RoboDK station: main for aircraft (copy).rdk

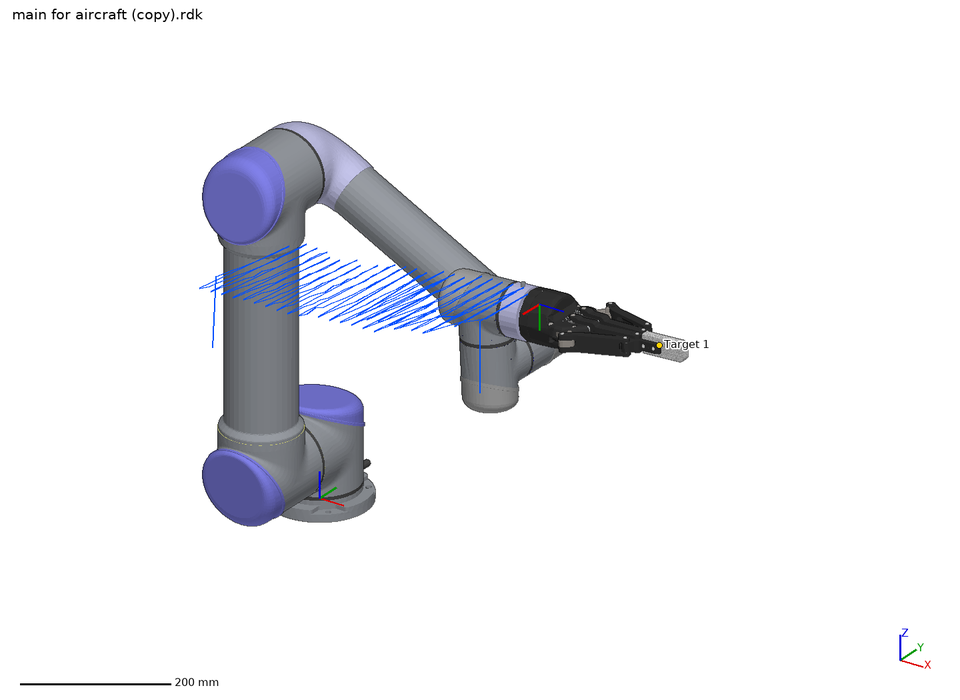
[picture v0: the station drawn from its stored meshes, robots at their saved joint values, targets as dots, program paths as lines]
Station main. Poses are relative to the parent item; angles as X-Y-Z fixed-axis rotations.
  - frame UR5 Base at (0, 0, 0) mm
    - robot UR5: 6 axes, payload 5 kg, reach 850 mm, repeatability 0.1 mm, weight 18.4 kg
        modified DH rows (alpha deg, a mm, theta deg, d mm): 0, 0, 0, 89.2; 90, 0, 180, 0; 0, 425, 0, 0; 0, 392.43, 0, 109; -90, 0, 0, 93.65; 90, 0, 180, 82
        joint limits [-360, -360, -360, -360, -360, -360] to [360, 360, 360, 360, 360, 360]; home [0, -90, -90, 0, 90, 0]; saved at [-0.013, -90.021, -116.97, 29.935, 90.025, 0.152]
      - tool RobotiQ 2-Finger-140 Closed, TCP at (0, 0, 200) mm, size 124 x 75 x 244.3 mm
    - target Target 1 (Cartesian target) at (626.33, -109, 443.99) mm, rotated rx -87.03 ry 0 rz -90 deg; joints [0, -90, -117.03, 30, 90, 0] of UR5
  - frame Object at (435.27, -113.47, 453.26) mm, rotated rx -90 ry 0 rz -90 deg
    - object cloud_1 at (0, 0, 0) mm
  - machining project Path1 settings: rotZ(0) | rotX(0)*rotY(0) | rotz(0) | onStart | onPathStart | onApproach | onPoint | onRetract | onFinish | SetRPM(%1) | SetTool(%1) | Extruder(%1) | default | default | OutOnMov(%1) | OutOffMov(%1) | onPathFinish | M_RunCode(%1)
  - program Path1 (311 instructions, listed below)
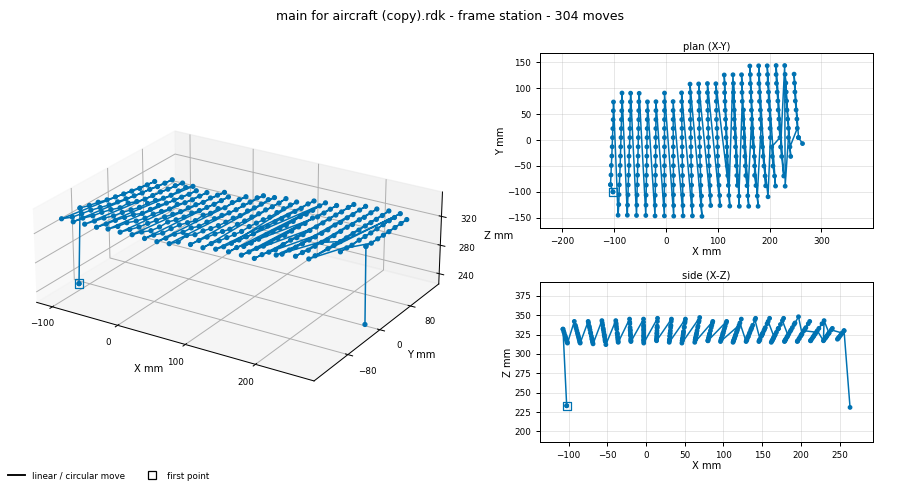
[picture p0: tool path of main for aircraft (copy).rdk in frame station, 304 of 304 moves have a stored position in this frame; points joined in program order, loops and branches not executed]

--- program Path1 (robot UR5) ---
  Smooth(10)
  Set Ref.: UR5 Base
  Set Tool: RobotiQ 2-Finger-140 Closed
  Show RobotiQ 2-Finger-140 Closed
  Set speed (1000.0 mm/s)
  MoveJ 1 to (-102.38, -99.99, 233.07) mm, rotated rx 0 ry 8.41 rz 109.19 deg; joints [12.602, -85.858, -96.132, -6.063, 80.274, 110.751]
  MoveL 2 to (-102.38, -99.99, 233.07) mm, rotated rx 0 ry 8.41 rz 109.19 deg; joints [12.602, -85.858, -96.132, -6.063, 80.274, 110.751]
  MoveL 3 to (-107.19, -86.18, 332) mm, rotated rx 0 ry 8.41 rz 109.19 deg; joints [10.562, -99.693, -83.593, -4.724, 82.295, 110.463]
  MoveL 4 to (-107.19, -86.18, 332) mm, rotated rx 0 ry 8.41 rz 109.19 deg; joints [10.562, -99.693, -83.593, -4.724, 82.295, 110.463]
  Set speed (25.0 mm/s)
  MoveL 5 to (-106.22, -67.34, 329) mm, rotated rx 0 ry 8.74 rz 104.18 deg; joints [10.87, -99.349, -86.354, -2.871, 81.384, 105.634]
  MoveL 6 to (-105.57, -48.98, 327) mm, rotated rx 0 ry 8.16 rz 105.57 deg; joints [10.82, -99.525, -89.316, 0.897, 81.464, 106.907]
  MoveL 7 to (-104.6, -30.75, 324) mm, rotated rx 0 ry 7.53 rz 107.19 deg; joints [10.76, -99.737, -92.273, 4.74, 81.545, 108.407]
  MoveL 8 to (-103.96, -12.89, 322) mm, rotated rx 0 ry 7.37 rz 117.72 deg; joints [10.016, -100.321, -94.773, 8.532, 83.469, 118.664]
  MoveL 9 to (-103.31, 4.75, 320) mm, rotated rx 0 ry 7.46 rz 117.73 deg; joints [9.953, -100.71, -96.926, 10.993, 83.577, 118.674]
  MoveL 10 to (-102.67, 22.18, 318) mm, rotated rx 0 ry 7.52 rz 128.57 deg; joints [9.186, -101.609, -99.093, 14.811, 85.544, 129.274]
  MoveL 11 to (-102.02, 39.38, 316) mm, rotated rx 0 ry 6.96 rz 132.96 deg; joints [9.121, -102.574, -101.234, 18.709, 85.65, 133.56]
  MoveL 12 to (-101.7, 56.55, 315) mm, rotated rx 0 ry 6.41 rz 138.18 deg; joints [9.085, -103.834, -103.068, 22.622, 85.712, 138.679]
  MoveL 13 to (-101.37, 73.6, 314) mm, rotated rx 0 ry 3.46 rz 132.88 deg; joints [10.558, -105.526, -105.133, 28.096, 81.808, 133.3]
  MoveL 14 to (-92.54, -145.08, 342) mm, rotated rx 0 ry 12.08 rz 94.29 deg; joints [9.643, -101.198, -70.072, -20.918, 81.468, 96.221]
  MoveL 15 to (-91.18, -124.47, 337) mm, rotated rx 0 ry 10.91 rz 107.25 deg; joints [8.275, -100.357, -75.36, -14.733, 85.077, 108.45]
  MoveL 16 to (-90.64, -105.34, 335) mm, rotated rx 0 ry 8.32 rz 121.32 deg; joints [7.646, -100.444, -80.524, -6.143, 86.725, 121.995]
  MoveL 17 to (-90.1, -86.44, 333) mm, rotated rx 0 ry 8.35 rz 111.38 deg; joints [8.357, -100.028, -83.281, -4.497, 84.755, 112.306]
  MoveL 18 to (-89.29, -67.55, 330) mm, rotated rx 0 ry 9.44 rz 103.06 deg; joints [8.831, -99.489, -85.62, -4.149, 83.408, 104.309]
  MoveL 19 to (-88.48, -48.98, 327) mm, rotated rx 0 ry 7.86 rz 110.36 deg; joints [8.456, -99.825, -89.329, 1.751, 84.342, 111.271]
  MoveL 20 to (-87.94, -30.85, 325) mm, rotated rx 0 ry 7.28 rz 107.7 deg; joints [8.741, -100.08, -92.048, 5.148, 83.531, 108.625]
  MoveL 21 to (-87.4, -12.93, 323) mm, rotated rx 0 ry 8.39 rz 105.46 deg; joints [8.687, -100.038, -93.905, 5.809, 83.628, 106.526]
  MoveL 22 to (-86.86, 4.77, 321) mm, rotated rx 0 ry 6.63 rz 99.81 deg; joints [9.338, -100.841, -96.822, 11.062, 81.85, 100.818]
  MoveL 23 to (-86.31, 22.25, 319) mm, rotated rx 0 ry 5.26 rz 109.06 deg; joints [8.973, -102.005, -99.329, 16.325, 82.775, 109.764]
  MoveL 24 to (-86.04, 39.63, 318) mm, rotated rx 0 ry 5.54 rz 114.92 deg; joints [8.583, -102.815, -101.017, 18.776, 83.783, 115.571]
  MoveL 25 to (-85.5, 56.73, 316) mm, rotated rx 0 ry 5.08 rz 117.6 deg; joints [8.547, -103.81, -102.937, 22.22, 83.831, 118.178]
  MoveL 26 to (-85.23, 73.83, 315) mm, rotated rx 0 ry 3.41 rz 99.66 deg; joints [9.627, -105.263, -104.828, 26.693, 80.961, 100.21]
  MoveL 27 to (-84.96, 90.83, 314) mm, rotated rx 0 ry 3.94 rz 89.7 deg; joints [9.971, -106.042, -106.185, 28.226, 80.032, 90.395]
  MoveL 28 to (-74.66, -145.08, 342) mm, rotated rx 0 ry 10.54 rz 100.52 deg; joints [7.023, -101.454, -71.046, -17.903, 85.006, 101.612]
  MoveL 29 to (-74.22, -125.57, 340) mm, rotated rx 0 ry 9.71 rz 108.2 deg; joints [6.378, -101.067, -75.24, -12.926, 86.723, 108.974]
  MoveL 30 to (-73.35, -105.66, 336) mm, rotated rx 0 ry 8.84 rz 106.92 deg; joints [6.599, -100.447, -79.464, -8.567, 86.038, 107.705]
  MoveL 31 to (-72.91, -86.7, 334) mm, rotated rx 0 ry 8.21 rz 101.06 deg; joints [7.161, -100.199, -82.829, -5.067, 84.48, 101.952]
  MoveL 32 to (-72.26, -67.75, 331) mm, rotated rx 0 ry 9.2 rz 96.58 deg; joints [7.42, -99.749, -85.325, -4.123, 83.725, 97.683]
  MoveL 33 to (-71.39, -48.98, 327) mm, rotated rx 0 ry 7.88 rz 97.73 deg; joints [7.389, -99.789, -89.038, 0.969, 83.737, 98.667]
  MoveL 34 to (-71.39, -31.04, 327) mm, rotated rx 0 ry 6.46 rz 99.7 deg; joints [7.385, -100.613, -91.81, 6.015, 83.747, 100.462]
  MoveL 35 to (-70.51, -12.93, 323) mm, rotated rx 0 ry 7.59 rz 98.3 deg; joints [7.329, -100.32, -94.011, 6.781, 83.826, 99.186]
  MoveL 36 to (-69.86, 4.75, 320) mm, rotated rx 0 ry 7.15 rz 99.07 deg; joints [7.281, -100.728, -96.551, 10.182, 83.898, 99.896]
  MoveL 37 to (-69.64, 22.25, 319) mm, rotated rx 0 ry 5.47 rz 89.8 deg; joints [7.973, -101.873, -99.092, 15.437, 82.044, 90.568]
  MoveL 38 to (-69.42, 39.63, 318) mm, rotated rx 0 ry 4.41 rz 89.88 deg; joints [7.965, -103.107, -101.143, 19.794, 82.05, 90.502]
  MoveL 39 to (-68.98, 56.73, 316) mm, rotated rx 0 ry 3.93 rz 98.35 deg; joints [7.596, -104.158, -102.988, 23.224, 82.992, 98.85]
  MoveL 40 to (-68.77, 73.83, 315) mm, rotated rx 0 ry 5.61 rz 89.69 deg; joints [7.94, -104.282, -104.219, 22.835, 82.068, 90.473]
  MoveL 41 to (-68.33, 90.54, 313) mm, rotated rx 0 ry 5.55 rz 74.23 deg; joints [8.823, -105.26, -105.973, 25.806, 79.709, 75.129]
  MoveL 42 to (-56.95, -145.51, 343) mm, rotated rx 0 ry 9.64 rz 101.74 deg; joints [4.945, -101.92, -71.114, -16.416, 87.075, 102.389]
  MoveL 43 to (-56.45, -125.57, 340) mm, rotated rx 0 ry 8.37 rz 100.44 deg; joints [5.18, -101.276, -75.726, -11.245, 86.385, 101.075]
  MoveL 44 to (-55.95, -105.97, 337) mm, rotated rx 0 ry 8.97 rz 99.84 deg; joints [5.141, -100.723, -78.806, -9.321, 86.447, 100.511]
  MoveL 45 to (-55.29, -86.44, 333) mm, rotated rx 0 ry 8.77 rz 103.79 deg; joints [4.782, -100.34, -82.357, -5.829, 87.353, 104.341]
  MoveL 46 to (-54.96, -67.75, 331) mm, rotated rx 0 ry 10.15 rz 95.9 deg; joints [5.361, -99.868, -84.468, -5.787, 85.759, 96.747]
  MoveL 47 to (-54.46, -49.13, 328) mm, rotated rx 0 ry 8.29 rz 89.76 deg; joints [5.984, -99.98, -88.428, 0.073, 84.044, 90.628]
  MoveL 48 to (-53.96, -30.85, 325) mm, rotated rx 0 ry 5.34 rz 95.68 deg; joints [5.649, -100.888, -92.308, 7.865, 84.903, 96.178]
  MoveL 49 to (-53.8, -12.97, 324) mm, rotated rx 0 ry 7.69 rz 102.43 deg; joints [4.957, -100.783, -93.45, 6.716, 86.735, 102.97]
  MoveL 50 to (-53.46, 4.78, 322) mm, rotated rx 0 ry 8.12 rz 110.5 deg; joints [4.228, -101.283, -95.457, 9.135, 88.645, 110.872]
  MoveL 51 to (-52.97, 22.25, 319) mm, rotated rx 0 ry 6.28 rz 105.85 deg; joints [4.88, -102.068, -98.402, 14.419, 86.859, 106.271]
  MoveL 52 to (-52.63, 39.51, 317) mm, rotated rx 0 ry 5.01 rz 96.55 deg; joints [5.559, -103.021, -100.779, 18.808, 85.033, 97.01]
  MoveL 53 to (-52.63, 56.9, 317) mm, rotated rx 0 ry 3.88 rz 89.83 deg; joints [5.917, -104.494, -102.589, 23.18, 84.085, 90.228]
  MoveL 54 to (-52.47, 74.07, 316) mm, rotated rx 0 ry 6.25 rz 89.29 deg; joints [5.936, -104.353, -103.631, 21.699, 84.022, 89.941]
  MoveL 55 to (-51.8, 90.26, 312) mm, rotated rx 0 ry 6.86 rz 83.81 deg; joints [6.305, -104.639, -105.472, 23.236, 83.002, 84.609]
  MoveL 56 to (-39.02, -145.51, 343) mm, rotated rx 0 ry 10.41 rz 100.77 deg; joints [2.876, -102.295, -70.06, -17.872, 89.105, 101.109]
  MoveL 57 to (-38.68, -125.57, 340) mm, rotated rx 0 ry 8.6 rz 107.1 deg; joints [2.527, -101.795, -75.104, -11.321, 90.02, 107.285]
  MoveL 58 to (-38.45, -106.28, 338) mm, rotated rx 0 ry 9.51 rz 102.38 deg; joints [2.79, -101.253, -77.786, -10.244, 89.276, 102.667]
  MoveL 59 to (-38.11, -86.96, 335) mm, rotated rx 0 ry 10.02 rz 98.86 deg; joints [3.049, -100.721, -80.786, -8.4, 88.533, 99.253]
  MoveL 60 to (-37.77, -67.95, 332) mm, rotated rx 0 ry 8.81 rz 100.35 deg; joints [3.01, -100.662, -84.566, -3.438, 88.601, 100.688]
  MoveL 61 to (-37.2, -48.98, 327) mm, rotated rx 0 ry 8.58 rz 104.58 deg; joints [2.636, -100.453, -87.878, 0.03, 89.545, 104.809]
  MoveL 62 to (-37.09, -30.94, 326) mm, rotated rx 0 ry 6.73 rz 109.13 deg; joints [2.605, -101.258, -91.051, 5.948, 89.613, 109.295]
  MoveL 63 to (-36.97, -13.01, 325) mm, rotated rx 0 ry 5.81 rz 112.71 deg; joints [2.578, -102.029, -93.568, 10.238, 89.673, 112.841]
  MoveL 64 to (-36.63, 4.78, 322) mm, rotated rx 0 ry 7.75 rz 102.62 deg; joints [2.874, -101.51, -95.208, 9.15, 88.841, 102.888]
  MoveL 65 to (-36.4, 22.32, 320) mm, rotated rx 0 ry 8.53 rz 105.62 deg; joints [2.497, -101.848, -96.972, 10.603, 89.819, 105.812]
  MoveL 66 to (-36.18, 39.63, 318) mm, rotated rx 0 ry 5.1 rz 103.06 deg; joints [3.176, -103.547, -100.132, 18.704, 87.988, 103.282]
  MoveL 67 to (-35.95, 56.73, 316) mm, rotated rx 0 ry 3.37 rz 99.81 deg; joints [3.515, -104.997, -102.361, 24.03, 87.065, 100.001]
  MoveL 68 to (-35.84, 73.83, 315) mm, rotated rx 0 ry 6.51 rz 97.07 deg; joints [3.362, -104.518, -103.198, 21.245, 87.46, 97.408]
  MoveL 69 to (-21.21, -146.36, 345) mm, rotated rx 0 ry 10.78 rz 100.32 deg; joints [0.831, -103.07, -68.684, -18.857, 91.104, 100.296]
  MoveL 70 to (-20.97, -125.94, 341) mm, rotated rx 0 ry 9.17 rz 96.23 deg; joints [1.341, -102.102, -74.004, -13.009, 89.667, 96.363]
  MoveL 71 to (-20.85, -106.6, 339) mm, rotated rx 0 ry 8.79 rz 89.96 deg; joints [1.903, -101.608, -77.676, -9.513, 88.113, 90.252]
  MoveL 72 to (-20.54, -86.7, 334) mm, rotated rx 0 ry 9.41 rz 86.82 deg; joints [2.181, -100.816, -81.091, -7.498, 87.329, 87.221]
  MoveL 73 to (-20.35, -67.75, 331) mm, rotated rx 0 ry 8.78 rz 100.37 deg; joints [0.958, -100.98, -84.233, -3.424, 90.627, 100.391]
  MoveL 74 to (-20.29, -49.43, 330) mm, rotated rx 0 ry 8.07 rz 105.51 deg; joints [0.619, -101.412, -87.053, 0.689, 91.538, 105.446]
  MoveL 75 to (-20.11, -31.04, 327) mm, rotated rx 0 ry 7.55 rz 102.54 deg; joints [0.903, -101.463, -90.018, 4.108, 90.74, 102.548]
  MoveL 76 to (-19.92, -12.97, 324) mm, rotated rx 0 ry 5.89 rz 95.38 deg; joints [1.529, -101.925, -93.313, 9.371, 89.03, 95.508]
  MoveL 77 to (-19.92, 4.81, 324) mm, rotated rx 0 ry 6.5 rz 94.93 deg; joints [1.525, -102.397, -94.965, 10.889, 89.042, 95.07]
  MoveL 78 to (-19.68, 22.32, 320) mm, rotated rx 0 ry 8.26 rz 97.94 deg; joints [1.159, -102.119, -96.662, 10.596, 89.991, 98.024]
  MoveL 79 to (-19.55, 39.63, 318) mm, rotated rx 0 ry 5.79 rz 107.49 deg; joints [0.794, -103.81, -99.357, 17.649, 90.946, 107.486]
  MoveL 80 to (-19.49, 56.9, 317) mm, rotated rx 0 ry 4.26 rz 114.24 deg; joints [0.782, -105.413, -101.378, 22.905, 90.968, 114.234]
  MoveL 81 to (-19.43, 74.07, 316) mm, rotated rx 0 ry 6.19 rz 111.98 deg; joints [0.436, -105.6, -102.418, 22.278, 91.878, 111.909]
  MoveL 82 to (-3.18, -146.36, 345) mm, rotated rx 0 ry 10.73 rz 100.34 deg; joints [-1.217, -103.634, -68.014, -18.926, 93.112, 99.939]
  MoveL 83 to (-3.14, -125.94, 341) mm, rotated rx 0 ry 11.27 rz 87.5 deg; joints [0.124, -102.309, -72.137, -16.813, 89.389, 87.57]
  MoveL 84 to (-3.11, -105.97, 337) mm, rotated rx 0 ry 10.22 rz 84.32 deg; joints [0.416, -101.559, -76.799, -11.811, 88.584, 84.481]
  MoveL 85 to (-3.09, -86.96, 335) mm, rotated rx 0 ry 7.59 rz 89.98 deg; joints [-0.16, -101.783, -81.227, -4.58, 90.156, 89.964]
  MoveL 86 to (-3.06, -67.95, 332) mm, rotated rx 0 ry 6.84 rz 103.6 deg; joints [-1.091, -102.038, -84.402, -0.215, 92.689, 103.379]
  MoveL 87 to (-3.04, -49.43, 330) mm, rotated rx 0 ry 8.39 rz 101.11 deg; joints [-1.099, -101.741, -86.307, -0.189, 92.699, 100.838]
  MoveL 88 to (-3.02, -31.04, 327) mm, rotated rx 0 ry 8.41 rz 97.48 deg; joints [-0.808, -101.633, -89.075, 2.362, 91.892, 97.288]
  MoveL 89 to (-2.99, -12.97, 324) mm, rotated rx 0 ry 5.88 rz 95.42 deg; joints [-0.504, -102.411, -92.718, 9.27, 91.056, 95.345]
  MoveL 90 to (-2.98, 4.8, 323) mm, rotated rx 0 ry 6.56 rz 99.89 deg; joints [-0.84, -102.841, -94.416, 10.789, 91.959, 99.728]
  MoveL 91 to (-2.96, 22.39, 321) mm, rotated rx 0 ry 8.19 rz 93.99 deg; joints [-0.516, -102.65, -96.025, 10.506, 91.08, 93.88]
  MoveL 92 to (-2.93, 39.63, 318) mm, rotated rx 0 ry 5.24 rz 109.31 deg; joints [-1.217, -104.536, -98.879, 18.461, 92.944, 109.132]
  MoveL 93 to (-2.93, 57.08, 318) mm, rotated rx 0 ry 3.75 rz 117.73 deg; joints [-1.224, -106.292, -100.706, 23.678, 92.964, 117.61]
  MoveL 94 to (-2.91, 74.07, 316) mm, rotated rx 0 ry 6.01 rz 107.04 deg; joints [-1.238, -105.986, -101.901, 22.137, 92.989, 106.829]
  MoveL 95 to (-2.9, 90.83, 314) mm, rotated rx 0 ry 8.15 rz 102.6 deg; joints [-1.251, -105.83, -103.026, 20.892, 93.012, 102.305]
  MoveL 96 to (14.9, -146.78, 346) mm, rotated rx 0 ry 10.58 rz 92.62 deg; joints [-2.457, -104.157, -67.286, -19.135, 92.897, 92.127]
  MoveL 97 to (14.72, -126.31, 342) mm, rotated rx 0 ry 12.07 rz 92.33 deg; joints [-2.453, -103.205, -70.364, -18.509, 92.886, 91.762]
  MoveL 98 to (14.46, -105.66, 336) mm, rotated rx 0 ry 9.79 rz 96.03 deg; joints [-2.767, -102.37, -76.175, -11.209, 93.75, 95.474]
  MoveL 99 to (14.38, -86.7, 334) mm, rotated rx 0 ry 5.33 rz 107.43 deg; joints [-3.109, -103.006, -81.616, -0.482, 94.692, 107.084]
  MoveL 100 to (14.38, -68.36, 334) mm, rotated rx 0 ry 7.78 rz 101.88 deg; joints [-3.102, -102.698, -82.806, -2.135, 94.671, 101.358]
  MoveL 101 to (14.21, -49.43, 330) mm, rotated rx 0 ry 10.19 rz 93.02 deg; joints [-2.489, -101.744, -84.835, -3.612, 92.983, 92.529]
  MoveL 102 to (14.08, -31.04, 327) mm, rotated rx 0 ry 6.92 rz 99.29 deg; joints [-2.837, -102.609, -89.019, 4.782, 93.932, 98.889]
  MoveL 103 to (14.03, -13.05, 326) mm, rotated rx 0 ry 5.97 rz 100.93 deg; joints [-2.85, -103.327, -91.556, 9.006, 93.966, 100.585]
  MoveL 104 to (13.91, 4.8, 323) mm, rotated rx 0 ry 7.02 rz 113.7 deg; joints [-3.826, -103.748, -93.3, 10.576, 96.619, 113.114]
  MoveL 105 to (13.82, 22.39, 321) mm, rotated rx 0 ry 7.7 rz 98.65 deg; joints [-2.862, -103.489, -95.404, 11.26, 93.991, 98.193]
  MoveL 106 to (13.73, 39.76, 319) mm, rotated rx 0 ry 5.75 rz 107.77 deg; joints [-3.221, -105.003, -97.866, 17.369, 94.961, 107.382]
  MoveL 107 to (13.69, 57.08, 318) mm, rotated rx 0 ry 2.98 rz 112.99 deg; joints [-2.883, -107.001, -100.217, 24.465, 94.045, 112.829]
  MoveL 108 to (13.65, 74.3, 317) mm, rotated rx 0 ry 6.62 rz 105.49 deg; joints [-3.227, -106.368, -100.895, 20.859, 94.971, 105.028]
  MoveL 109 to (32.89, -146.36, 345) mm, rotated rx 0 ry 10.2 rz 84.56 deg; joints [-3.687, -104.429, -67.314, -18.421, 92.668, 83.997]
  MoveL 110 to (32.6, -126.31, 342) mm, rotated rx 0 ry 10.93 rz 97.86 deg; joints [-5.021, -104.126, -70.137, -16.631, 96.418, 96.776]
  MoveL 111 to (32.12, -105.97, 337) mm, rotated rx 0 ry 10.44 rz 104.05 deg; joints [-5.594, -103.496, -74.436, -12.293, 98.027, 102.836]
  MoveL 112 to (32.03, -87.21, 336) mm, rotated rx 0 ry 6.19 rz 115.52 deg; joints [-5.706, -104.098, -79.801, -1.745, 98.342, 114.83]
  MoveL 113 to (31.84, -68.36, 334) mm, rotated rx 0 ry 8.14 rz 90.15 deg; joints [-4.215, -102.954, -82.094, -3.115, 94.194, 89.555]
  MoveL 114 to (31.46, -49.43, 330) mm, rotated rx 0 ry 10.66 rz 90.09 deg; joints [-4.184, -102.205, -83.905, -4.578, 94.128, 89.311]
  MoveL 115 to (31.07, -30.94, 326) mm, rotated rx 0 ry 5.28 rz 90.17 deg; joints [-4.205, -103.361, -89.271, 7.34, 94.203, 89.78]
  MoveL 116 to (31.17, -13.09, 327) mm, rotated rx 0 ry 5.96 rz 100.94 deg; joints [-4.841, -104.101, -90.583, 8.806, 95.944, 100.391]
  MoveL 117 to (30.79, 4.8, 323) mm, rotated rx 0 ry 7.52 rz 94.41 deg; joints [-4.51, -103.579, -92.684, 8.734, 95.047, 93.779]
  MoveL 118 to (30.79, 22.53, 323) mm, rotated rx 0 ry 7.63 rz 94.41 deg; joints [-4.514, -104.263, -94.441, 11.066, 95.059, 93.771]
  MoveL 119 to (30.31, 39.63, 318) mm, rotated rx 0 ry 4.96 rz 97.03 deg; joints [-4.531, -105.491, -97.649, 18.192, 95.121, 96.615]
  MoveL 120 to (30.41, 57.26, 319) mm, rotated rx 0 ry 2.81 rz 102.12 deg; joints [-4.529, -107.619, -99.406, 24.271, 95.112, 101.892]
  MoveL 121 to (30.22, 74.3, 317) mm, rotated rx 0 ry 5.15 rz 108.57 deg; joints [-5.128, -107.635, -100.424, 23.145, 96.747, 108.059]
  MoveL 122 to (30.03, 91.12, 315) mm, rotated rx 0 ry 5.56 rz 104.8 deg; joints [-4.997, -108.236, -101.985, 24.81, 96.393, 104.259]
  MoveL 123 to (50.92, -146.36, 345) mm, rotated rx 0 ry 11.06 rz 97.54 deg; joints [-6.983, -105.741, -65.013, -20.323, 98.297, 96.066]
  MoveL 124 to (50.48, -126.31, 342) mm, rotated rx 0 ry 8.95 rz 113.5 deg; joints [-8.14, -105.608, -70.208, -12.561, 101.613, 112.059]
  MoveL 125 to (50.18, -106.91, 340) mm, rotated rx 0 ry 9.24 rz 106.56 deg; joints [-7.631, -104.869, -73.51, -10.617, 100.162, 105.167]
  MoveL 126 to (49.44, -86.96, 335) mm, rotated rx 0 ry 9.48 rz 109.47 deg; joints [-7.906, -104.284, -77.111, -7.702, 100.955, 107.979]
  MoveL 127 to (49.3, -68.36, 334) mm, rotated rx 0 ry 9.07 rz 90.13 deg; joints [-6.19, -103.51, -80.707, -4.901, 96.133, 89.151]
  MoveL 128 to (48.56, -49.28, 329) mm, rotated rx 0 ry 10.66 rz 92.94 deg; joints [-6.443, -102.892, -83.087, -4.742, 96.874, 91.692]
  MoveL 129 to (48.41, -31.13, 328) mm, rotated rx 0 ry 5.83 rz 84.78 deg; joints [-5.878, -104.048, -87.973, 6.189, 95.318, 84.213]
  MoveL 130 to (48.12, -13.05, 326) mm, rotated rx 0 ry 5.33 rz 90.21 deg; joints [-6.182, -104.609, -90.334, 9.58, 96.174, 89.632]
  MoveL 131 to (47.82, 4.81, 324) mm, rotated rx 0 ry 7.2 rz 76.49 deg; joints [-5.193, -104.12, -92.385, 9.49, 93.476, 75.959]
  MoveL 132 to (47.38, 22.39, 321) mm, rotated rx 0 ry 7.14 rz 99.47 deg; joints [-6.803, -105.001, -93.912, 11.801, 97.924, 98.562]
  MoveL 133 to (47.08, 39.76, 319) mm, rotated rx 0 ry 4.41 rz 97.99 deg; joints [-6.495, -106.524, -96.747, 18.87, 97.088, 97.467]
  MoveL 134 to (47.08, 57.26, 319) mm, rotated rx 0 ry 4.01 rz 125.33 deg; joints [-7.472, -108.39, -97.913, 22.981, 99.779, 124.828]
  MoveL 135 to (46.79, 74.3, 317) mm, rotated rx 0 ry 4.5 rz 121.3 deg; joints [-7.475, -108.943, -99.475, 24.517, 99.794, 120.718]
  MoveL 136 to (46.79, 91.7, 317) mm, rotated rx 0 ry 6.11 rz 121.36 deg; joints [-7.941, -109.626, -100.266, 24.578, 101.082, 120.479]
  MoveL 137 to (46.34, 108.07, 314) mm, rotated rx 0 ry 10.92 rz 117.12 deg; joints [-8.885, -108.695, -100.471, 19.168, 103.71, 115.154]
  MoveL 138 to (69.35, -147.2, 347) mm, rotated rx 0 ry 12 rz 99.79 deg; joints [-9.237, -107.157, -62.368, -22.52, 101.064, 97.663]
  MoveL 139 to (68.15, -125.94, 341) mm, rotated rx 0 ry 7.89 rz 98 deg; joints [-8.776, -105.727, -70.4, -11.805, 99.788, 96.716]
  MoveL 140 to (68.55, -107.86, 343) mm, rotated rx 0 ry 8.48 rz 97.55 deg; joints [-8.787, -105.837, -72.46, -10.235, 99.802, 96.168]
  MoveL 141 to (67.15, -87.21, 336) mm, rotated rx 0 ry 10.36 rz 95.98 deg; joints [-8.708, -104.568, -75.681, -10.205, 99.64, 94.313]
  MoveL 142 to (66.75, -68.36, 334) mm, rotated rx 0 ry 9.61 rz 99.51 deg; joints [-8.982, -104.614, -79.001, -6.02, 100.437, 97.877]
  MoveL 143 to (65.96, -49.43, 330) mm, rotated rx 0 ry 10.69 rz 87.23 deg; joints [-7.801, -103.571, -82.191, -5, 97.153, 85.83]
  MoveL 144 to (65.36, -31.04, 327) mm, rotated rx 0 ry 6.34 rz 85.26 deg; joints [-7.823, -104.524, -86.994, 5.147, 97.253, 84.424]
  MoveL 145 to (64.96, -13.01, 325) mm, rotated rx 0 ry 4.93 rz 77.04 deg; joints [-7.493, -105.162, -90.026, 10.35, 96.361, 76.456]
  MoveL 146 to (64.76, 4.81, 324) mm, rotated rx 0 ry 6.51 rz 100.09 deg; joints [-8.728, -105.642, -90.876, 10.01, 99.812, 99.041]
  MoveL 147 to (64.16, 22.39, 321) mm, rotated rx 0 ry 6.34 rz 111.08 deg; joints [-9.349, -106.434, -92.917, 13.312, 101.575, 109.985]
  MoveL 148 to (64.16, 40, 321) mm, rotated rx 0 ry 4.74 rz 127.04 deg; joints [-9.682, -108.313, -94.835, 19.275, 102.513, 126.291]
  MoveL 149 to (63.76, 57.26, 319) mm, rotated rx 0 ry 4.94 rz 117.85 deg; joints [-9.37, -108.619, -96.702, 20.86, 101.649, 117.032]
  MoveL 150 to (63.56, 74.54, 318) mm, rotated rx 0 ry 3.5 rz 109.62 deg; joints [-8.739, -109.8, -98.764, 25.22, 99.899, 109.083]
  MoveL 151 to (63.56, 91.99, 318) mm, rotated rx 0 ry 4.51 rz 121.63 deg; joints [-9.402, -110.978, -99.543, 26.596, 101.746, 120.908]
  MoveL 152 to (62.96, 108.41, 315) mm, rotated rx 0 ry 7.19 rz 112.07 deg; joints [-9.55, -110.437, -100.692, 24.312, 102.18, 110.779]
  MoveL 153 to (86.23, -126.31, 342) mm, rotated rx 0 ry 9.23 rz 87.58 deg; joints [-9.907, -106.325, -68.517, -14.504, 99.39, 86.01]
  MoveL 154 to (85.73, -106.91, 340) mm, rotated rx 0 ry 8.04 rz 83.22 deg; joints [-9.609, -105.849, -72.899, -9.328, 98.569, 81.939]
  MoveL 155 to (84.97, -87.47, 337) mm, rotated rx 0 ry 11.02 rz 79.42 deg; joints [-8.967, -104.812, -74.94, -11.158, 96.794, 77.915]
  MoveL 156 to (84.21, -68.36, 334) mm, rotated rx 0 ry 9.54 rz 86.91 deg; joints [-9.768, -104.966, -78.512, -6.174, 99.12, 85.324]
  MoveL 157 to (83.2, -49.43, 330) mm, rotated rx 0 ry 10.68 rz 87.2 deg; joints [-9.71, -104.409, -81.138, -5.255, 99.022, 85.435]
  MoveL 158 to (82.2, -30.94, 326) mm, rotated rx 0 ry 6.38 rz 100.32 deg; joints [-10.641, -105.636, -85.603, 4.824, 101.718, 99.078]
  MoveL 159 to (82.2, -13.05, 326) mm, rotated rx 0 ry 4.07 rz 114.45 deg; joints [-10.957, -107.168, -88.228, 11.6, 102.617, 113.674]
  MoveL 160 to (81.69, 4.81, 324) mm, rotated rx 0 ry 6.45 rz 115.59 deg; joints [-11.516, -107.114, -89.394, 10.509, 104.236, 114.256]
  MoveL 161 to (81.44, 22.53, 323) mm, rotated rx 0 ry 6.04 rz 101.08 deg; joints [-10.632, -107.237, -91.86, 13.044, 101.733, 99.9]
  MoveL 162 to (80.94, 40, 321) mm, rotated rx 0 ry 4.5 rz 105.14 deg; joints [-10.641, -108.452, -94.195, 18.21, 101.785, 104.278]
  MoveL 163 to (80.68, 57.44, 320) mm, rotated rx 0 ry 3.88 rz 98.82 deg; joints [-10.319, -109.369, -96.124, 21.587, 100.89, 98.097]
  MoveL 164 to (80.18, 74.54, 318) mm, rotated rx 0 ry 3.49 rz 109.56 deg; joints [-10.624, -110.562, -97.682, 24.884, 101.774, 108.904]
  MoveL 165 to (79.93, 91.7, 317) mm, rotated rx 0 ry 4.04 rz 107.19 deg; joints [-10.627, -111.304, -99.005, 26.365, 101.796, 106.425]
  MoveL 166 to (79.93, 109.1, 317) mm, rotated rx 0 ry 5.62 rz 99.39 deg; joints [-10.459, -111.611, -100.069, 26.021, 101.325, 98.319]
  MoveL 167 to (104.11, -126.31, 342) mm, rotated rx 0 ry 10.94 rz 100.97 deg; joints [-13.037, -107.98, -65.179, -17.951, 104.871, 98.279]
  MoveL 168 to (103.5, -106.91, 340) mm, rotated rx 0 ry 9.27 rz 99.63 deg; joints [-12.788, -107.383, -70.024, -12.017, 104.166, 97.434]
  MoveL 169 to (102.28, -87.21, 336) mm, rotated rx 0 ry 9.33 rz 90.07 deg; joints [-11.956, -106.273, -74.217, -9.042, 101.807, 88.107]
  MoveL 170 to (101.37, -68.16, 333) mm, rotated rx 0 ry 9.49 rz 93.26 deg; joints [-12.199, -106.038, -77.195, -6.476, 102.567, 91.173]
  MoveL 171 to (100.45, -49.43, 330) mm, rotated rx 0 ry 10.2 rz 99.03 deg; joints [-12.712, -105.992, -79.546, -4.85, 104.105, 96.619]
  MoveL 172 to (99.54, -31.04, 327) mm, rotated rx 0 ry 5.74 rz 125.49 deg; joints [-13.675, -107.821, -83.922, 6.86, 106.955, 124.198]
  MoveL 173 to (99.54, -13.09, 327) mm, rotated rx 0 ry 4.97 rz 132.47 deg; joints [-13.696, -108.728, -86.154, 11.054, 107.017, 131.458]
  MoveL 174 to (98.93, 4.83, 325) mm, rotated rx 0 ry 6.9 rz 113.84 deg; joints [-13.359, -107.994, -87.831, 9.256, 106.06, 112.169]
  MoveL 175 to (98.32, 22.53, 323) mm, rotated rx 0 ry 6.13 rz 106.2 deg; joints [-12.783, -108.274, -90.488, 12.68, 104.422, 104.766]
  MoveL 176 to (97.41, 39.88, 320) mm, rotated rx 0 ry 5.55 rz 102.18 deg; joints [-12.475, -108.717, -92.953, 16.091, 103.586, 100.919]
  MoveL 177 to (97.41, 57.44, 320) mm, rotated rx 0 ry 3.99 rz 107.03 deg; joints [-12.49, -110.353, -94.753, 21.177, 103.631, 106.146]
  MoveL 178 to (97.11, 74.77, 319) mm, rotated rx 0 ry 4.46 rz 97.66 deg; joints [-12.165, -110.834, -96.397, 22.702, 102.722, 96.682]
  MoveL 179 to (96.8, 91.99, 318) mm, rotated rx 0 ry 3.37 rz 100.37 deg; joints [-12.171, -112.38, -97.941, 26.926, 102.756, 99.638]
  MoveL 180 to (96.19, 108.76, 316) mm, rotated rx 0 ry 3.39 rz 85.16 deg; joints [-11.662, -113.085, -99.707, 29.348, 101.356, 84.474]
  MoveL 181 to (120.2, -87.47, 337) mm, rotated rx 0 ry 11.39 rz 105.6 deg; joints [-15.3, -108.21, -70.373, -12.959, 108.052, 102.274]
  MoveL 182 to (119.13, -68.36, 334) mm, rotated rx 0 ry 8.68 rz 103.94 deg; joints [-14.852, -107.855, -75.561, -5.379, 106.769, 101.537]
  MoveL 183 to (118.06, -49.58, 331) mm, rotated rx 0 ry 8.38 rz 116.28 deg; joints [-15.651, -108.359, -78.321, -1.27, 109.209, 113.895]
  MoveL 184 to (116.99, -31.13, 328) mm, rotated rx 0 ry 5.99 rz 129.64 deg; joints [-15.731, -109.161, -82.141, 6.411, 109.496, 128.161]
  MoveL 185 to (117.35, -13.17, 329) mm, rotated rx 0 ry 6.18 rz 122.8 deg; joints [-15.494, -109.48, -83.951, 7.947, 108.77, 121.18]
  MoveL 186 to (115.92, 4.83, 325) mm, rotated rx 0 ry 7.5 rz 98.76 deg; joints [-14.298, -108.114, -86.823, 7.253, 105.314, 96.792]
  MoveL 187 to (115.56, 22.6, 324) mm, rotated rx 0 ry 6.64 rz 104.97 deg; joints [-14.6, -109.163, -88.875, 11.362, 106.217, 103.195]
  MoveL 188 to (114.85, 40.13, 322) mm, rotated rx 0 ry 4.87 rz 118.31 deg; joints [-14.916, -110.711, -91.114, 17.337, 107.18, 117.068]
  MoveL 189 to (114.14, 57.44, 320) mm, rotated rx 0 ry 4.43 rz 121.51 deg; joints [-14.904, -111.592, -93.019, 20.662, 107.183, 120.421]
  MoveL 190 to (113.78, 74.77, 319) mm, rotated rx 0 ry 5.09 rz 103.56 deg; joints [-14.296, -111.615, -94.835, 21.32, 105.432, 102.239]
  MoveL 191 to (113.07, 91.7, 317) mm, rotated rx 0 ry 3.5 rz 109.84 deg; joints [-14.288, -113.241, -96.629, 26.455, 105.451, 108.962]
  MoveL 192 to (113.07, 109.1, 317) mm, rotated rx 0 ry 4.26 rz 114.74 deg; joints [-14.595, -114.318, -97.475, 27.766, 106.341, 113.667]
  MoveL 193 to (112.35, 125.7, 315) mm, rotated rx 0 ry 7.55 rz 117.68 deg; joints [-15.435, -114.292, -97.909, 25.136, 108.827, 115.597]
  MoveL 194 to (123.05, -127.42, 345) mm, rotated rx 0 ry 11.81 rz 113.8 deg; joints [-16.182, -110.57, -61.425, -19.552, 110.617, 110.137]
  MoveL 195 to (121.27, -106.91, 340) mm, rotated rx 0 ry 11.54 rz 112.57 deg; joints [-15.993, -109.32, -66.269, -15.757, 110.107, 109.046]
  MoveL 196 to (129.23, 126.1, 316) mm, rotated rx 0 ry 5.68 rz 99.25 deg; joints [-15.877, -115.167, -97.586, 26.898, 106.71, 97.609]
  MoveL 197 to (137.82, -87.47, 337) mm, rotated rx 0 ry 11.64 rz 100.27 deg; joints [-16.58, -108.988, -68.958, -14.124, 108.298, 96.638]
  MoveL 198 to (136.59, -68.36, 334) mm, rotated rx 0 ry 9.05 rz 100.11 deg; joints [-16.378, -108.715, -74.038, -6.602, 107.755, 97.363]
  MoveL 199 to (135.77, -49.73, 332) mm, rotated rx 0 ry 6.81 rz 103.97 deg; joints [-16.429, -109.141, -77.917, 0.108, 107.957, 101.918]
  MoveL 200 to (135.36, -31.42, 331) mm, rotated rx 0 ry 5.77 rz 96.28 deg; joints [-15.925, -109.29, -81.076, 4.382, 106.474, 94.613]
  MoveL 201 to (134.14, -13.13, 328) mm, rotated rx 0 ry 6.36 rz 95.8 deg; joints [-15.883, -109.175, -83.515, 6.096, 106.425, 93.966]
  MoveL 202 to (133.32, 4.84, 326) mm, rotated rx 0 ry 6.4 rz 90.57 deg; joints [-15.561, -109.279, -86.018, 8.652, 105.525, 88.79]
  MoveL 203 to (132.09, 22.53, 323) mm, rotated rx 0 ry 5.59 rz 107.75 deg; joints [-16.373, -110.422, -87.967, 12.792, 108.002, 106.099]
  MoveL 204 to (131.68, 40.13, 322) mm, rotated rx 0 ry 4.65 rz 137.21 deg; joints [-17.243, -112.537, -89.394, 18.557, 110.627, 136.114]
  MoveL 205 to (131.68, 57.8, 322) mm, rotated rx 0 ry 6.11 rz 118.91 deg; joints [-16.989, -112.347, -90.716, 17.375, 109.863, 117.114]
  MoveL 206 to (130.46, 74.77, 319) mm, rotated rx 0 ry 7.67 rz 112.69 deg; joints [-16.928, -112.121, -92.349, 16.954, 109.744, 110.322]
  MoveL 207 to (130.05, 91.99, 318) mm, rotated rx 0 ry 2.81 rz 102.37 deg; joints [-15.773, -114.406, -95.386, 26.931, 106.356, 101.576]
  MoveL 208 to (130.05, 109.44, 318) mm, rotated rx 0 ry 3.52 rz 109.9 deg; joints [-16.076, -115.489, -96.216, 28.242, 107.245, 108.905]
  MoveL 209 to (141.5, -127.79, 346) mm, rotated rx 0 ry 10.32 rz 93.34 deg; joints [-16.004, -110.526, -61.821, -18.394, 106.336, 90.337]
  MoveL 210 to (140.68, -108.17, 344) mm, rotated rx 0 ry 11.45 rz 102.65 deg; joints [-16.871, -110.479, -64.107, -17.234, 109.029, 98.999]
  MoveL 211 to (147.13, 74.77, 319) mm, rotated rx 0 ry 6.65 rz 96.13 deg; joints [-17.53, -112.637, -91.979, 17.657, 108.118, 93.998]
  MoveL 212 to (146.67, 91.99, 318) mm, rotated rx 0 ry 3.35 rz 100.46 deg; joints [-17.51, -115.073, -93.907, 25.509, 108.089, 99.399]
  MoveL 213 to (146.21, 109.1, 317) mm, rotated rx 0 ry 3.37 rz 100.47 deg; joints [-17.497, -116.096, -95.205, 27.811, 108.079, 99.399]
  MoveL 214 to (145.75, 126.1, 316) mm, rotated rx 0 ry 3.75 rz 88.77 deg; joints [-17.123, -116.782, -96.691, 29.551, 107.005, 87.619]
  MoveL 215 to (156.35, -87.99, 339) mm, rotated rx 0 ry 13.38 rz 88.06 deg; joints [-17.078, -109.569, -66.643, -17.722, 106.153, 84.058]
  MoveL 216 to (154.05, -68.36, 334) mm, rotated rx 0 ry 8.55 rz 94.22 deg; joints [-17.668, -109.633, -73.076, -6.267, 108.093, 91.462]
  MoveL 217 to (153.13, -49.73, 332) mm, rotated rx 0 ry 4.18 rz 98.06 deg; joints [-17.695, -110.605, -77.758, 4.009, 108.232, 96.72]
  MoveL 218 to (152.2, -31.32, 330) mm, rotated rx 0 ry 7.3 rz 99.02 deg; joints [-17.891, -110.007, -78.999, 1.389, 108.884, 96.609]
  MoveL 219 to (150.82, -13.09, 327) mm, rotated rx 0 ry 8.39 rz 90.43 deg; joints [-17.29, -109.325, -81.736, 2.274, 107.162, 87.822]
  MoveL 220 to (150.36, 4.84, 326) mm, rotated rx 0 ry 5.87 rz 90.49 deg; joints [-17.317, -110.509, -84.728, 9.091, 107.274, 88.66]
  MoveL 221 to (149.9, 22.67, 325) mm, rotated rx 0 ry 5.39 rz 90.53 deg; joints [-17.309, -111.226, -86.808, 12.388, 107.28, 88.846]
  MoveL 222 to (148.97, 40.25, 323) mm, rotated rx 0 ry 2.68 rz 92.94 deg; joints [-17.353, -112.896, -89.271, 19.358, 107.471, 92.103]
  MoveL 223 to (149.44, 58.16, 324) mm, rotated rx 0 ry 4.9 rz 92 deg; joints [-17.362, -113.005, -90.18, 18.05, 107.467, 90.462]
  MoveL 224 to (159.58, -127.79, 346) mm, rotated rx 0 ry 9.43 rz 90.48 deg; joints [-17.551, -111.667, -60.894, -17.322, 107.384, 87.502]
  MoveL 225 to (157.74, -107.54, 342) mm, rotated rx 0 ry 11.34 rz 90.34 deg; joints [-17.437, -110.555, -63.965, -17.357, 107.153, 86.799]
  MoveL 226 to (165.34, 40.13, 322) mm, rotated rx 0 ry 3.98 rz 55.89 deg; joints [-17.854, -112.831, -88.859, 18.266, 105.591, 54.904]
  MoveL 227 to (164.83, 57.62, 321) mm, rotated rx 0 ry 5.23 rz 72.13 deg; joints [-18.135, -113.042, -89.979, 17.832, 106.462, 70.587]
  MoveL 228 to (164.32, 75.01, 320) mm, rotated rx 0 ry 6.12 rz 85.86 deg; joints [-18.68, -113.694, -90.883, 18.158, 108.13, 83.828]
  MoveL 229 to (163.8, 92.28, 319) mm, rotated rx 0 ry 3.91 rz 99.04 deg; joints [-19.219, -115.945, -92.149, 23.988, 109.787, 97.671]
  MoveL 230 to (162.78, 109.1, 317) mm, rotated rx 0 ry 3.51 rz 109.84 deg; joints [-19.475, -117.249, -93.412, 27.136, 110.631, 108.635]
  MoveL 231 to (162.78, 126.5, 317) mm, rotated rx 0 ry 2.79 rz 111.34 deg; joints [-19.395, -118.817, -94.506, 30.556, 110.387, 110.4]
  MoveL 232 to (161.75, 142.99, 315) mm, rotated rx 0 ry 5.34 rz 113.35 deg; joints [-19.874, -118.873, -95.271, 28.86, 111.911, 111.463]
  MoveL 233 to (173.56, -87.73, 338) mm, rotated rx 0 ry 12.03 rz 108.38 deg; joints [-20.799, -112.333, -64.304, -15.878, 114.124, 103.577]
  MoveL 234 to (170.99, -68.16, 333) mm, rotated rx 0 ry 9.46 rz 112.83 deg; joints [-20.768, -111.782, -69.983, -7.788, 114.164, 109.166]
  MoveL 235 to (170.99, -49.88, 333) mm, rotated rx 0 ry 7.09 rz 122.31 deg; joints [-20.889, -112.621, -73.518, -0.45, 114.551, 119.765]
  MoveL 236 to (170.48, -31.51, 332) mm, rotated rx 0 ry 8.03 rz 109.51 deg; joints [-20.333, -111.943, -75.998, -0.268, 112.817, 106.482]
  MoveL 237 to (168.43, -13.13, 328) mm, rotated rx 0 ry 8.43 rz 101.46 deg; joints [-19.79, -111.182, -79.259, 1.575, 111.243, 98.349]
  MoveL 238 to (166.89, 4.83, 325) mm, rotated rx 0 ry 5.87 rz 96.02 deg; joints [-19.288, -111.661, -83.129, 8.586, 109.798, 93.941]
  MoveL 239 to (166.37, 22.6, 324) mm, rotated rx 0 ry 5.56 rz 78.42 deg; joints [-18.428, -111.785, -85.963, 12.05, 107.229, 76.671]
  MoveL 240 to (177.67, -127.79, 346) mm, rotated rx 0 ry 10.14 rz 125.61 deg; joints [-21.909, -115.54, -56.206, -17.547, 117.545, 121.711]
  MoveL 241 to (176.13, -107.86, 343) mm, rotated rx 0 ry 11.44 rz 113.11 deg; joints [-21.198, -113.812, -59.923, -17.907, 115.277, 108.498]
  MoveL 242 to (183.31, 22.6, 324) mm, rotated rx 0 ry 5.24 rz 115.3 deg; joints [-21.707, -114.31, -82.859, 11.99, 113.864, 113.295]
  MoveL 243 to (182.18, 40.13, 322) mm, rotated rx 0 ry 4.63 rz 127.23 deg; joints [-21.949, -115.404, -84.759, 16.107, 114.699, 125.621]
  MoveL 244 to (182.18, 57.8, 322) mm, rotated rx 0 ry 5.34 rz 115.88 deg; joints [-21.716, -115.612, -86.327, 16.68, 113.964, 113.84]
  MoveL 245 to (180.48, 74.77, 319) mm, rotated rx 0 ry 4.67 rz 112.45 deg; joints [-21.419, -116.117, -88.655, 20.078, 113.137, 110.673]
  MoveL 246 to (180.48, 92.28, 319) mm, rotated rx 0 ry 4.46 rz 98.37 deg; joints [-20.88, -116.738, -90.471, 22.472, 111.463, 96.659]
  MoveL 247 to (179.35, 109.1, 317) mm, rotated rx 0 ry 3.92 rz 99.61 deg; joints [-20.853, -117.817, -92.036, 25.703, 111.457, 98.115]
  MoveL 248 to (179.35, 126.5, 317) mm, rotated rx 0 ry 2.28 rz 105.51 deg; joints [-20.849, -119.906, -93.069, 30.611, 111.443, 104.657]
  MoveL 249 to (178.78, 143.44, 316) mm, rotated rx 0 ry 4.57 rz 101.36 deg; joints [-20.945, -119.884, -94.068, 29.127, 111.777, 99.604]
  MoveL 250 to (192.36, -88.25, 340) mm, rotated rx 0 ry 14.31 rz 118.57 deg; joints [-23.679, -115.36, -58.963, -20.17, 119.83, 112.012]
  MoveL 251 to (191.23, -69.18, 338) mm, rotated rx 0 ry 10.5 rz 121.78 deg; joints [-23.252, -114.723, -65.469, -9.953, 118.445, 117.34]
  MoveL 252 to (188.97, -50.03, 334) mm, rotated rx 0 ry 8.34 rz 117.24 deg; joints [-22.51, -113.757, -70.803, -3.699, 116.113, 113.834]
  MoveL 253 to (187.27, -31.42, 331) mm, rotated rx 0 ry 7.3 rz 102.92 deg; joints [-21.494, -112.784, -75.16, 0.215, 112.946, 99.991]
  MoveL 254 to (186.14, -13.17, 329) mm, rotated rx 0 ry 9.38 rz 100.13 deg; joints [-21.413, -112.288, -76.948, -0.786, 112.762, 96.354]
  MoveL 255 to (184.44, 4.84, 326) mm, rotated rx 0 ry 7.61 rz 107.06 deg; joints [-21.685, -113.077, -80.003, 5.128, 113.726, 103.986]
  MoveL 256 to (196.89, -109.43, 348) mm, rotated rx 0 ry 8.54 rz 102.79 deg; joints [-21.844, -115.311, -59.185, -14.586, 113.482, 99.287]
  MoveL 257 to (201.48, 4.84, 326) mm, rotated rx 0 ry 7.7 rz 110.81 deg; joints [-23.502, -114.548, -77.926, 4.457, 116.03, 107.442]
  MoveL 258 to (200.86, 22.67, 325) mm, rotated rx 0 ry 5.99 rz 129.41 deg; joints [-24.007, -116.339, -79.94, 11.053, 117.72, 127.128]
  MoveL 259 to (200.24, 40.38, 324) mm, rotated rx 0 ry 4.92 rz 132.26 deg; joints [-23.791, -117.136, -82.215, 15.261, 117.047, 130.5]
  MoveL 260 to (199.63, 57.98, 323) mm, rotated rx 0 ry 6.53 rz 126.76 deg; joints [-24.009, -117.35, -83.376, 14.815, 117.801, 124.172]
  MoveL 261 to (197.77, 75.01, 320) mm, rotated rx 0 ry 5.59 rz 120.97 deg; joints [-23.514, -117.582, -86.054, 18.291, 116.298, 118.718]
  MoveL 262 to (197.77, 92.57, 320) mm, rotated rx 0 ry 5.64 rz 120.99 deg; joints [-23.526, -118.565, -87.308, 20.475, 116.337, 118.709]
  MoveL 263 to (195.92, 109.1, 317) mm, rotated rx 0 ry 4.57 rz 105.53 deg; joints [-22.715, -118.796, -90.022, 24.003, 113.865, 103.623]
  MoveL 264 to (195.92, 126.5, 317) mm, rotated rx 0 ry 2.01 rz 125.62 deg; joints [-22.719, -121.432, -91.032, 30.677, 113.879, 124.908]
  MoveL 265 to (195.3, 143.44, 316) mm, rotated rx 1.22 ry -0.93 rz -91.24 deg; joints [-22.716, -122.957, -92.016, 33.93, 113.911, 268.359]
  MoveL 266 to (211.37, -88.77, 342) mm, rotated rx 0 ry 12.2 rz 97.41 deg; joints [-23.104, -114.994, -59.803, -18.48, 114.117, 92.067]
  MoveL 267 to (209.51, -69.39, 339) mm, rotated rx 0 ry 10.52 rz 105.86 deg; joints [-23.686, -115.034, -64.083, -12.165, 116.146, 101.095]
  MoveL 268 to (206.42, -50.03, 334) mm, rotated rx 0 ry 10.07 rz 104.62 deg; joints [-23.475, -114.127, -68.51, -8.179, 115.639, 100.116]
  MoveL 269 to (205.19, -31.51, 332) mm, rotated rx 0 ry 7.38 rz 106.88 deg; joints [-23.346, -114.476, -72.748, -0.59, 115.293, 103.661]
  MoveL 270 to (203.95, -13.21, 330) mm, rotated rx 0 ry 8.53 rz 108.32 deg; joints [-23.52, -114.435, -74.721, 0.144, 115.938, 104.538]
  MoveL 271 to (219.86, 4.87, 328) mm, rotated rx 0 ry 7.08 rz 108.65 deg; joints [-24.889, -116.176, -75.906, 4.554, 116.963, 105.356]
  MoveL 272 to (218.52, 22.74, 326) mm, rotated rx 0 ry 4.28 rz 121.49 deg; joints [-24.898, -117.57, -78.842, 12.312, 117.078, 119.69]
  MoveL 273 to (217.85, 40.5, 325) mm, rotated rx 0 ry 5.06 rz 109.6 deg; joints [-24.628, -117.476, -80.841, 13.004, 116.23, 107.317]
  MoveL 274 to (216.51, 57.98, 323) mm, rotated rx 0 ry 5.62 rz 107.91 deg; joints [-24.592, -117.722, -82.714, 14.478, 116.2, 105.348]
  MoveL 275 to (215.84, 75.48, 322) mm, rotated rx 0 ry 4.64 rz 112.08 deg; joints [-24.598, -118.922, -84.439, 18.569, 116.265, 110.021]
  MoveL 276 to (214.5, 92.57, 320) mm, rotated rx 0 ry 5.88 rz 125.54 deg; joints [-25.279, -119.96, -85.138, 19.651, 118.595, 123.067]
  MoveL 277 to (213.16, 109.44, 318) mm, rotated rx 0 ry 5.65 rz 120.81 deg; joints [-25.017, -120.446, -87.043, 21.999, 117.812, 118.365]
  MoveL 278 to (212.49, 126.5, 317) mm, rotated rx 0 ry 3.93 rz 137.09 deg; joints [-25.021, -122.546, -88.276, 27.798, 117.868, 135.747]
  MoveL 279 to (212.49, 143.9, 317) mm, rotated rx 1.7 ry -0.97 rz -91.73 deg; joints [-24.499, -124.301, -89.714, 32.876, 116.162, 267.8]
  MoveL 280 to (227.23, -69.39, 339) mm, rotated rx 0 ry 10.15 rz 116.92 deg; joints [-25.972, -117.497, -61.238, -11.737, 120.185, 111.974]
  MoveL 281 to (223.21, -31.61, 333) mm, rotated rx 0 ry 9.64 rz 112.64 deg; joints [-25.522, -116.23, -68.766, -5.169, 118.878, 107.986]
  MoveL 282 to (221.2, -13.21, 330) mm, rotated rx 0 ry 8.83 rz 100.82 deg; joints [-24.611, -115.235, -73.113, -1.308, 115.959, 96.687]
  MoveL 283 to (229.06, 143.9, 317) mm, rotated rx 0 ry 2.37 rz 137.25 deg; joints [-26.03, -125.108, -87.8, 31.089, 117.76, 136.425]
  MoveL 284 to (229.92, -89.03, 343) mm, rotated rx 0 ry 10.45 rz 100.9 deg; joints [-24.931, -117.073, -58.089, -16.313, 116.464, 95.914]
  MoveL 285 to (236.28, 4.86, 327) mm, rotated rx 0 ry 7.18 rz 112.56 deg; joints [-26.579, -117.614, -73.803, 3.828, 119.129, 109.007]
  MoveL 286 to (236.28, 22.81, 327) mm, rotated rx 0 ry 5.19 rz 115.82 deg; joints [-26.417, -118.69, -76.35, 9.717, 118.58, 113.362]
  MoveL 287 to (234.84, 40.5, 325) mm, rotated rx 0 ry 5.54 rz 107.68 deg; joints [-26.122, -118.57, -78.758, 11.362, 117.682, 104.978]
  MoveL 288 to (233.39, 57.98, 323) mm, rotated rx 0 ry 5.49 rz 102.08 deg; joints [-25.851, -118.766, -81.077, 13.82, 116.876, 99.406]
  MoveL 289 to (232.67, 75.48, 322) mm, rotated rx 0 ry 4.47 rz 104.9 deg; joints [-25.849, -119.933, -82.822, 17.904, 116.918, 102.739]
  MoveL 290 to (231.95, 92.86, 321) mm, rotated rx 0 ry 4.66 rz 112.11 deg; joints [-26.087, -120.957, -83.964, 20.044, 117.757, 109.896]
  MoveL 291 to (231.22, 110.13, 320) mm, rotated rx 0 ry 5.15 rz 123.63 deg; joints [-26.534, -122.249, -84.68, 22.008, 119.304, 121.322]
  MoveL 292 to (229.78, 126.9, 318) mm, rotated rx 0 ry 4.3 rz 131.65 deg; joints [-26.513, -123.584, -86.136, 26.032, 119.325, 129.925]
  MoveL 293 to (240.62, -31.61, 333) mm, rotated rx 0 ry 10.88 rz 103.15 deg; joints [-26.452, -116.814, -66.6, -8.654, 118.417, 97.574]
  MoveL 294 to (239.17, -13.25, 331) mm, rotated rx 0 ry 8.01 rz 109.77 deg; joints [-26.612, -117.576, -70.485, -0.565, 119.059, 105.736]
  MoveL 295 to (253.38, 22.81, 327) mm, rotated rx 0 ry 6.33 rz 134.45 deg; joints [-28.74, -121.11, -72.696, 8.414, 123.069, 131.681]
  MoveL 296 to (252.6, 40.63, 326) mm, rotated rx 0 ry 5.94 rz 112.14 deg; joints [-27.829, -120.248, -75.996, 9.899, 119.921, 109.076]
  MoveL 297 to (251.05, 58.16, 324) mm, rotated rx 0 ry 6 rz 112.15 deg; joints [-27.796, -120.623, -78.045, 12.26, 119.908, 109.052]
  MoveL 298 to (249.5, 75.48, 322) mm, rotated rx 0 ry 4.21 rz 106.3 deg; joints [-27.336, -121.36, -80.764, 17.523, 118.443, 104.143]
  MoveL 299 to (248.73, 92.86, 321) mm, rotated rx 0 ry 3.3 rz 89.96 deg; joints [-26.822, -122.054, -83.006, 21.36, 116.772, 88.288]
  MoveL 300 to (247.95, 110.13, 320) mm, rotated rx 0 ry 4.27 rz 106.16 deg; joints [-27.294, -122.962, -83.657, 21.952, 118.405, 103.979]
  MoveL 301 to (247.18, 127.3, 319) mm, rotated rx 0 ry 4.69 rz 119.73 deg; joints [-27.745, -124.323, -84.228, 23.851, 119.99, 117.46]
  MoveL 302 to (255.7, 4.9, 330) mm, rotated rx 0 ry 8.04 rz 123.54 deg; joints [-28.748, -120.326, -69.588, 1.93, 122.956, 119.442]
  Set speed (1000.0 mm/s)
  MoveL 303 to (255.7, 4.9, 330) mm, rotated rx 0 ry 8.04 rz 123.54 deg; joints [-28.748, -120.326, -69.588, 1.93, 122.956, 119.442]
  MoveL 304 to (263.43, -6.75, 230.98) mm, rotated rx 0 ry 8.04 rz 123.54 deg; joints [-34.537, -110.415, -82.427, 4.256, 128.684, 118.413]
